FUNCTION_BLOCK M_EL6_SERIAL IMPLEMENTS IFC_GENERIC_COMMUNICATION_INTERFACE
VAR_INPUT
END_VAR
VAR_OUTPUT
END_VAR
VAR
	//Hardware Buffers
		IN_Hardward_Buffer AT %I*	: EL6inData22B;
		OUT_Hardward_Buffer AT %Q*	: EL6outData22B;
		//IN_Hardward_Buffer AT %I*	: PcComInData;
		//OUT_Hardward_Buffer AT %Q* 	: PcComOutData;
	//Software Buffers
		_txBuffer : ComBuffer;
		_rxBuffer : ComBuffer;
	//Serial Properties
		_UsePrefix 	: BOOL := FALSE;
		_UseSuffix 	: BOOL := FALSE;
		_Prefix		: STRING(5);
		_Suffix		: STRING(5);
		_LineError	: BOOL := FALSE;
	//Serial FunctionBlocks
		M_RECEIVE	: ReceiveData;
		M_SEND		: SendData;
		M_SERIALCONTROLLER : SerialLineControl;
END_VAR

METHOD Close_Connection : ph_lv0.RETURN_CODE
Close_Connection := ph_lv0.LV0_RETURNCODE.RETURN_SUCCESS;
END_METHOD

METHOD Create_Handle : ph_lv0.RETURN_CODE
VAR_INPUT
	Configuration	: PH_LV1_GENERIC_COMMUNICATION_INTERFACE.S_GCI_CONFIG;
	OUT_HANDLE	: POINTER TO UDINT;
END_VAR
Create_Handle := ph_lv0.LV0_RETURNCODE.RETURN_SUCCESS;
END_METHOD

METHOD Hardware_Buffer_IO : Return_Code
VAR_INPUT
END_VAR
M_SERIALCONTROLLER(
	Mode:= SERIALLINEMODE_EL6_22B, 
	pComIn:= ADR(IN_Hardward_Buffer), 
	pComOut:= ADR(OUT_Hardward_Buffer), 
	SizeComIn:= SIZEOF(IN_Hardward_Buffer), 
	Error=> , 
	ErrorID=> , 
	TxBuffer:= _txBuffer, 
	RxBuffer:= _rxBuffer);
IF M_SERIALCONTROLLER.Error THEN
	_LineError := TRUE;
ELSE
	_LineError := FALSE;
END_IF
END_METHOD

METHOD Open_Connection : ph_lv0.RETURN_CODE
VAR_INPUT
	CONNECTION_INFO	: PH_LV1_GENERIC_COMMUNICATION_INTERFACE.S_GCI_CONFIG;
END_VAR
IF _LineError THEN
	Open_Connection := ph_lv0.LV0_RETURNCODE.RETURN_ERROR;
ELSE
	Open_Connection := ph_lv0.LV0_RETURNCODE.RETURN_SUCCESS;
END_IF
END_METHOD

PROPERTY Prefix : STRING(5)
GET
Prefix := _Prefix;
END_GET
SET
_Prefix := Prefix;
END_SET
END_PROPERTY

METHOD Read : ph_lv0.RETURN_CODE
VAR_INPUT
	Configuration	: PH_LV1_GENERIC_COMMUNICATION_INTERFACE.S_GCI_CONFIG;
END_VAR
IF _LineError THEN
	Read := ph_lv0.LV0_RETURNCODE.RETURN_ERROR;
ELSE
	IF _UsePrefix THEN
		M_RECEIVE.pPrefix := ADR(_Prefix);
		M_RECEIVE.LenPrefix := INT_TO_BYTE(LEN(_Prefix));
	ELSE
		M_RECEIVE.LenPrefix := 0;
	END_IF
	IF _UseSuffix THEN
		M_RECEIVE.pSuffix := ADR(_Suffix);
		M_RECEIVE.LenSuffix := INT_TO_BYTE(LEN(_Suffix));
	ELSE
		M_RECEIVE.LenSuffix := 0;
	END_IF
	M_RECEIVE(
		pReceiveData:= Configuration.P_Data, 
		SizeReceiveData:= Configuration.Data_Size, 
		RXbuffer:= _rxBuffer);
	IF M_RECEIVE.Error THEN
		Read := ph_lv0.LV0_RETURNCODE.RETURN_ERROR;
	ELSIF NOT _UseSuffix AND M_RECEIVE.RxTimeout THEN
		Read := ph_lv0.LV0_RETURNCODE.RETURN_SUCCESS;
	ELSIF NOT M_RECEIVE.busy THEN
		Read := ph_lv0.LV0_RETURNCODE.RETURN_SUCCESS;
	ELSE
		Read := ph_lv0.LV0_RETURNCODE.RETURN_BUSY;
	END_IF
END_IF
END_METHOD

METHOD Release_Handle : ph_lv0.RETURN_CODE
VAR_INPUT
	IN_HANDLE	: POINTER TO UDINT;
END_VAR
Release_Handle := ph_lv0.LV0_RETURNCODE.RETURN_SUCCESS;
END_METHOD

PROPERTY Serial_Line_Error : BOOL
GET
END_GET
SET
END_SET
END_PROPERTY

PROPERTY Suffix : STRING(5)
GET
Suffix := _Suffix;
END_GET
SET
_Suffix := Suffix;
END_SET
END_PROPERTY

PROPERTY Use_Prefix : BOOL
GET
Use_Prefix := _UsePrefix;
END_GET
SET
_UsePrefix := Use_Prefix;
END_SET
END_PROPERTY

PROPERTY Use_Suffix : BOOL
GET
Use_Suffix := _UseSuffix;
END_GET
SET
_UseSuffix := Use_Suffix;
END_SET
END_PROPERTY

METHOD Write : ph_lv0.RETURN_CODE
VAR_INPUT
	Configuration	: PH_LV1_GENERIC_COMMUNICATION_INTERFACE.S_GCI_CONFIG;
END_VAR
IF _LineError THEN
	Write := ph_lv0.LV0_RETURNCODE.RETURN_ERROR;
ELSE
	M_SEND(
		pSendData:= Configuration.P_Data, 
		Length:= Configuration.Data_Size, 
		Busy=> , 
		Error=> , 
		TXbuffer:= _txBuffer);
	IF M_SEND.Error THEN
		Write := ph_lv0.LV0_RETURNCODE.RETURN_ERROR;
	ELSIF NOT M_SEND.busy THEN
		Write := ph_lv0.LV0_RETURNCODE.RETURN_SUCCESS;
	ELSE
		Write := ph_lv0.LV0_RETURNCODE.RETURN_BUSY;
	END_IF
END_IF
END_METHOD

END_FUNCTION_BLOCK

(* stored: Version 1.1.0.1, ProductVersion 3.1.4019.2
   POU M_EL6_SERIAL: Id {d7913f93-3dbb-469e-9dc5-be0540c05df4}, SpecialFunc None
   Folder Methods: Id {4badb3e5-319a-4754-b5a9-44eb76f70dd4}
   Folder Generic Interface: Id {b84fa621-bb52-4ff0-859a-07b997acdcef}
   Method Close_Connection: Id {881a2dc3-c121-48dd-a1db-15f07fa7e94a}
   Method Create_Handle: Id {b6efaa31-fd9c-427b-9142-ed9eed5a5fcc}
   Method Hardware_Buffer_IO: Id {23764e00-2150-4f69-9fb8-32517259fcaf}
   Method Open_Connection: Id {7c75ab7a-cf3f-4c83-8f51-26ad48474f2c}
   Property Prefix: Id {26e32199-7889-4569-beaa-af633856625b}
   Get Get: Id {b7fd11f5-2d97-403e-a936-24f93fabf7dc}
   Set Set: Id {c752f0d5-bbc8-442e-a3ae-b727f8220f28}
   Method Read: Id {4f9acb4b-09fe-4919-8980-31f43b2b0aa6}
   Method Release_Handle: Id {fbc61870-a439-4017-93f5-814c6d613470}
   Property Serial_Line_Error: Id {fb9b637f-d021-45cf-8362-02e18a6080d3}
   Get Get: Id {4f5d208a-230a-4d6d-bf42-841ff8eb08ba}
   Set Set: Id {82605c86-f685-4ab1-8eaf-0ce6789c6be5}
   Property Suffix: Id {4465ef3b-3ca0-4db0-9ecc-2a9ee207cc14}
   Get Get: Id {0b8012fa-c158-4362-8d6d-82cec696a455}
   Set Set: Id {70f2830b-18dd-478e-ae7f-e64f4f77df39}
   Property Use_Prefix: Id {cc26f5d2-c764-417b-8c4a-37a516071961}
   Get Get: Id {9df5d8e3-46ea-4eca-ac02-1925336f4bdb}
   Set Set: Id {5ffadeb4-89a6-4eca-8124-aa788e5a31f4}
   Property Use_Suffix: Id {46598f32-dfbc-49b5-b617-24cb2f90c498}
   Get Get: Id {c5bc9b28-5230-4d96-9ff5-b2059ac2e4ba}
   Set Set: Id {96a0ff08-6a6c-4ef8-8279-2852241b39ae}
   Method Write: Id {b2ac8412-10c0-4097-bac9-99f5630bac28} *)
